(* CODESYS project IndraLogic.project

Project tree, tasks and I/O mapping:
  MLD : IndraDrive MLD-2G MPx20, Bosch Rexroth AG, order no. FWA-INDRV_-MPx-20VRS, version 20.24.1422.3503
    application Application
      task PlcTask (cyclic, interval t#20ms, priority 1) calls PlcProg, PlcProg
      program PlcProg [ST]
      global variables IO
    Parameter_IO : Drive I/O, Bosch Rexroth AG, version 20.1.2.0
        unmapped channels: Input P-0-1390, Input P-0-1391, Input P-0-1392, Input P-0-1393, Input P-0-1394, Input P-0-1395, Input P-0-1396, Input P-0-1397, Input P-0-1398, Input P-0-1399, Input P-0-1400, Input P-0-1401, Input P-0-1402, Input P-0-1403, Input P-0-1404, Input P-0-1405, Input P-0-1406, Input P-0-1407, Input P-0-1408, Input P-0-1409, Not Available, Not Available, Not Available, Not Available, Not Available, Not Available, Not Available, Not Available, Not Available, Not Available, Not Available, Not Available, Not Available, Not Available, Not Available, Input P-0-1440, Input P-0-1441, Input P-0-1442, Input P-0-1443, Input P-0-1444,
          Input P-0-1445, Input P-0-1446, Input P-0-1447, Output P-0-1410, Output P-0-1411, Output P-0-1412, Output P-0-1413, Output P-0-1414, Output P-0-1415, Output P-0-1416, Output P-0-1417, Output P-0-1418, Output P-0-1419, Output P-0-1420, Output P-0-1421, Output P-0-1422, Output P-0-1423, Output P-0-1424, Output P-0-1425, Output P-0-1426, Output P-0-1427, Output P-0-1428, Output P-0-1429
*)

// MLD/Application/IO
{attribute 'qualified_only'}
VAR_GLOBAL
	bEnableAxis AT %IX1.0 :BOOL;
	bExecuteVelocity AT %IX1.1 :BOOL;
	bChangeVelocity AT %IX1.2 :BOOL;
	bStopAxis AT %IX1.3 :BOOL;
END_VAR

// MLD/Application/PlcProg
PROGRAM PlcProg
VAR
	rVelocity :REAL;
	bIsAxisEnabled :BOOL;
	pwrOn: MC_Power;
	moveVel: MC_MoveVelocity;
	stopAxis: MC_Stop;
END_VAR

IF IO.bChangeVelocity THEN
	rVelocity := -20;
ELSE
	rVelocity := 100;
END_IF


pwrOn(
	Enable:= IO.bEnableAxis, 
	Status=> bIsAxisEnabled , 
	Error=> , 
	ErrorID=> , 
	ErrorIdent=> , 
	Axis:= Axis1 );
	
moveVel(
	Execute:= IO.bExecuteVelocity, 
	Velocity:= rVelocity , 
	Acceleration:= 1000, 
	Deceleration:= 1000 , 
	InVelocity=> , 
	Active=> , 
	CommandAborted=> , 
	Error=> , 
	ErrorID=> , 
	ErrorIdent=> , 
	Axis:= Axis1 );
	
stopAxis(
	Execute:= IO.bStopAxis , 
	Deceleration:= 1000 , 
	Done=> , 
	Active=> , 
	CommandAborted=> , 
	Error=> , 
	ErrorID=> , 
	ErrorIdent=> , 
	Axis:=Axis1 );

END_PROGRAM
